Universal Robots PolyScope program: Safe_Home_BeforeStart.urp

Program Safe_Home_BeforeStart (createdIn=3.2.18744 lastSavedIn=3.2.18744 directory=/home/ur/ursim-3.2/programs/Safe_home_pose installation=default robotSerialNumber=2014359999)
Calibrated DH parameters: a=[0, -0.425, -0.39225, 0, 0, 0]; d=[0.089159, 0, 0, 0.10915, 0.09465, 0.0823]; alpha=[1.570796, 0, 0, 1.570796, -1.570796, 0]; deltaTheta=[0, 0, 0, 0, 0, 0]
BeforeStart
  Folder Safe Home Folder
    'Read robot current position'
    start_pose := get_actual_tcp_pose()
    MoveL speed 250 mm/s, acceleration 1200 mm/s^2 (recalculateMotions=false) feature=Base
      'First pose is current pose'
      'Variable position'
      Waypoint Waypoint (Variable): variable=start_pose
    'Break start pose into directions'
    start_x := start_pose[0]
    start_y := start_pose[1]
    start_z := start_pose[2]
    'If TCP is inside box'
    If (start_x≥0.2) and (start_y≥0.1)
      'Move to safe pos. 50 mm above box edge'
      Safe_Z_value := 0.350
      'Same as start pose, but with altered Z-value'
      Safe_Pose := p[start_pose[0],start_pose[1],Safe_Z_value,start_pose[3],start_pose[4],start_pose[5]]
      MoveL speed 250 mm/s, acceleration 1200 mm/s^2 (recalculateMotions=false) feature=Base
        Waypoint Waypoint (Variable): variable=Safe_Pose
Robot Program (runOnlyOnce=false motionType=MoveJ speed=1.047198 acceleration=1.396263 recalculateMotions=false)
  MoveJ speed 60 deg/s, acceleration 80 deg/s^2 (recalculateMotions=false)
    Waypoint Normal_start: TCP in base x=-120.113 y=-431.763 z=221.664 mm, rx=-0.0012 ry=3.1163 rz=0.0389 rad; joints [-91.713, -91.336, -120.636, -59.501, 91.393, -1.776] deg
